// TIA Portal V20 export
DATA_BLOCK "DB_Global"   // DB23
// stored: Access Published, MemoryReserve 100, Namespace Global
   VAR
      Status : Struct
         Line : Struct
            ProductionLine : Struct
               On : Array[_.gminProductionLine.._.gmaxProductionLine] of Bool;
               ReadyToRun : Array[_.gminProductionLine.._.gmaxProductionLine] of Bool;
               Occupied : Array[_.gminProductionLine.._.gmaxProductionLine] of Bool;
               Running : Array[_.gminProductionLine.._.gmaxProductionLine] of Bool;
               Fault : Array[_.gminProductionLine.._.gmaxProductionLine] of Bool;
               Estop : Array[_.gminProductionLine.._.gmaxProductionLine] of Bool;
               Manual : Array[_.gminProductionLine.._.gmaxProductionLine] of Bool;
               Stop : Array[_.gminProductionLine.._.gmaxProductionLine] of Bool;
               Blockage : Array[_.gminProductionLine.._.gmaxProductionLine] of Bool;
            END_STRUCT;
            EmptyLine : Struct
               On : Array[_.gminEmptyLine.._.gmaxEmptyLine] of Bool;
               ReadyToRun : Array[_.gminEmptyLine.._.gmaxEmptyLine] of Bool;
               Occupied : Array[_.gminEmptyLine.._.gmaxEmptyLine] of Bool;
               Running : Array[_.gminEmptyLine.._.gmaxEmptyLine] of Bool;
               Fault : Array[_.gminEmptyLine.._.gmaxEmptyLine] of Bool;
               Estop : Array[_.gminEmptyLine.._.gmaxEmptyLine] of Bool;
               Manual : Array[_.gminEmptyLine.._.gmaxEmptyLine] of Bool;
               Stop : Array[_.gminEmptyLine.._.gmaxEmptyLine] of Bool;
               Blockage : Array[_.gminEmptyLine.._.gmaxEmptyLine] of Bool;
            END_STRUCT;
            PackedLine : Struct
               On : Array[_.gminPackedLine.._.gmaxPackedLine] of Bool;
               ReadyToRun : Array[_.gminPackedLine.._.gmaxPackedLine] of Bool;
               Occupied : Array[_.gminPackedLine.._.gmaxPackedLine] of Bool;
               Running : Array[_.gminPackedLine.._.gmaxPackedLine] of Bool;
               Fault : Array[_.gminPackedLine.._.gmaxPackedLine] of Bool;
               Estop : Array[_.gminPackedLine.._.gmaxPackedLine] of Bool;
               Manual : Array[_.gminPackedLine.._.gmaxPackedLine] of Bool;
               Stop : Array[_.gminPackedLine.._.gmaxPackedLine] of Bool;
               Blockage : Array[_.gminPackedLine.._.gmaxPackedLine] of Bool;
            END_STRUCT;
         END_STRUCT;
      END_STRUCT;
   END_VAR
BEGIN
   // Status.Line.ProductionLine.On[1001] : AS1.1.1
   // Status.Line.ProductionLine.On[1002] : AS1.1.2
   // Status.Line.ProductionLine.ReadyToRun[1001] : AS1.1.1
   // Status.Line.ProductionLine.ReadyToRun[1002] : AS1.1.2
   // Status.Line.ProductionLine.Occupied[1001] : AS1.1.1
   // Status.Line.ProductionLine.Occupied[1002] : AS1.1.2
   // Status.Line.ProductionLine.Running[1001] : AS1.1.1
   // Status.Line.ProductionLine.Running[1002] : AS1.1.2
   Status.Line.ProductionLine.Fault[1001] := 0;   // AS1.1.1
   Status.Line.ProductionLine.Fault[1002] := 0;   // AS1.1.2
   Status.Line.ProductionLine.Estop[1001] := 0;   // AS1.1.1
   Status.Line.ProductionLine.Estop[1002] := 0;   // AS1.1.2
   Status.Line.ProductionLine.Manual[1001] := 0;   // AS1.1.1
   Status.Line.ProductionLine.Manual[1002] := 0;   // AS1.1.2
   Status.Line.ProductionLine.Stop[1001] := 0;   // AS1.1.1
   Status.Line.ProductionLine.Stop[1002] := 0;   // AS1.1.2
   Status.Line.ProductionLine.Blockage[1001] := 0;   // AS1.1.1
   Status.Line.ProductionLine.Blockage[1002] := 0;   // AS1.1.2
   // Status.Line.PackedLine.ReadyToRun[3001] : BP1.1.1
   // Status.Line.PackedLine.ReadyToRun[3002] : BP1.1.2
   // Status.Line.PackedLine.Occupied[3001] : BP1.1.1
   // Status.Line.PackedLine.Occupied[3002] : BP1.1.2
   // Status.Line.PackedLine.Running[3001] : BP1.1.1
   // Status.Line.PackedLine.Running[3002] : BP1.1.2
   // Status.Line.PackedLine.Fault[3001] : BP1.1.1
   // Status.Line.PackedLine.Fault[3002] : BP1.1.2
   // Status.Line.PackedLine.Estop[3001] : BP1.1.1
   // Status.Line.PackedLine.Estop[3002] : BP1.1.2
   // Status.Line.PackedLine.Manual[3001] : BP1.1.1
   // Status.Line.PackedLine.Manual[3002] : BP1.1.2
   // Status.Line.PackedLine.Stop[3001] : BP1.1.1
   // Status.Line.PackedLine.Stop[3002] : BP1.1.2
   // Status.Line.PackedLine.Blockage[3001] : BP1.1.1
   // Status.Line.PackedLine.Blockage[3002] : BP1.1.2
END_DATA_BLOCK
